FUNCTION_BLOCK FB_CHP EXTENDS FB_ActorContinous
VAR_INPUT
END_VAR
VAR_OUTPUT
END_VAR
VAR
END_VAR

END_FUNCTION_BLOCK

(* stored: Version 1.1.0.1, ProductVersion 3.1.4024.10
   POU FB_CHP: Id {b646d58b-e895-49ef-8279-111f006d4387}, SpecialFunc None *)
